// TIA Portal V19 export
FUNCTION "RECIPE" : Void   // FC7, LAD
{ S7_Optimized_Access := 'TRUE' }
// stored: SetENOAutomatically false
BEGIN

REGION Network 1: RINSE 1
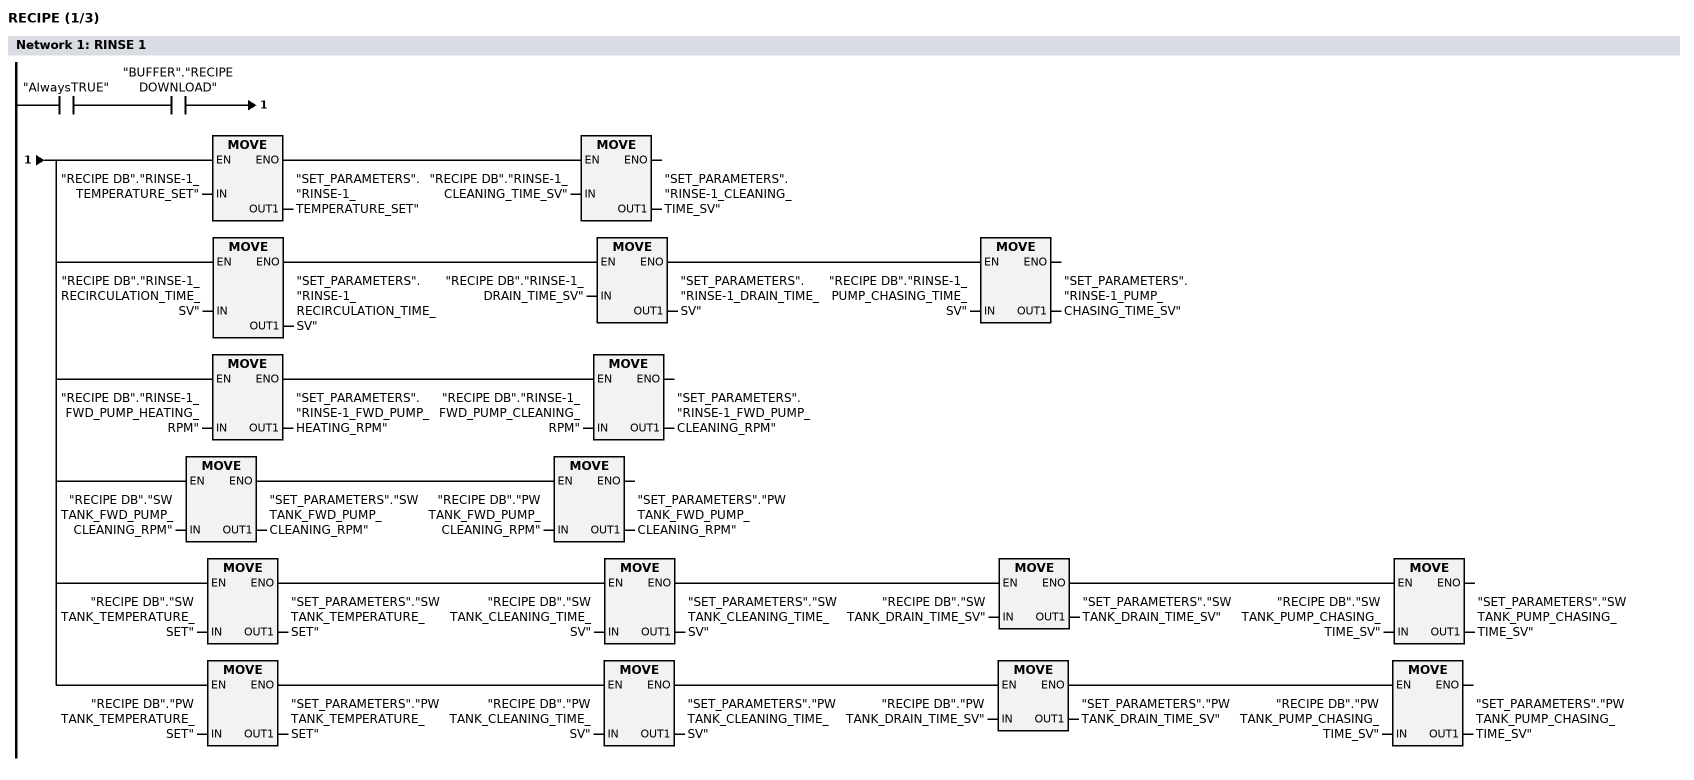
   RUNG wire#powerrail
      Contact( "AlwaysTRUE" )
      Contact( "BUFFER"."RECIPE DOWNLOAD" )
      wire#w1
      Move(in := "RECIPE DB"."RINSE-1_TEMPERATURE_SET", out1 => "SET_PARAMETERS"."RINSE-1_TEMPERATURE_SET")
      Move(in := "RECIPE DB"."RINSE-1_CLEANING_TIME_SV", out1 => "SET_PARAMETERS"."RINSE-1_CLEANING_TIME_SV")
   END_RUNG
   RUNG wire#w1
      Move(in := "RECIPE DB"."RINSE-1_RECIRCULATION_TIME_SV", out1 => "SET_PARAMETERS"."RINSE-1_RECIRCULATION_TIME_SV")
      Move(in := "RECIPE DB"."RINSE-1_DRAIN_TIME_SV", out1 => "SET_PARAMETERS"."RINSE-1_DRAIN_TIME_SV")
      Move(in := "RECIPE DB"."RINSE-1_PUMP_CHASING_TIME_SV", out1 => "SET_PARAMETERS"."RINSE-1_PUMP_CHASING_TIME_SV")
   END_RUNG
   RUNG wire#w1
      Move(in := "RECIPE DB"."RINSE-1_FWD_PUMP_HEATING_RPM", out1 => "SET_PARAMETERS"."RINSE-1_FWD_PUMP_HEATING_RPM")
      Move(in := "RECIPE DB"."RINSE-1_FWD_PUMP_CLEANING_RPM", out1 => "SET_PARAMETERS"."RINSE-1_FWD_PUMP_CLEANING_RPM")
   END_RUNG
   RUNG wire#w1
      Move(in := "RECIPE DB"."SW TANK_FWD_PUMP_CLEANING_RPM", out1 => "SET_PARAMETERS"."SW TANK_FWD_PUMP_CLEANING_RPM")
      Move(in := "RECIPE DB"."PW TANK_FWD_PUMP_CLEANING_RPM", out1 => "SET_PARAMETERS"."PW TANK_FWD_PUMP_CLEANING_RPM")
   END_RUNG
   RUNG wire#w1
      Move(in := "RECIPE DB"."SW TANK_TEMPERATURE_SET", out1 => "SET_PARAMETERS"."SW TANK_TEMPERATURE_SET")
      Move(in := "RECIPE DB"."SW TANK_CLEANING_TIME_SV", out1 => "SET_PARAMETERS"."SW TANK_CLEANING_TIME_SV")
      Move(in := "RECIPE DB"."SW TANK_DRAIN_TIME_SV", out1 => "SET_PARAMETERS"."SW TANK_DRAIN_TIME_SV")
      Move(in := "RECIPE DB"."SW TANK_PUMP_CHASING_TIME_SV", out1 => "SET_PARAMETERS"."SW TANK_PUMP_CHASING_TIME_SV")
   END_RUNG
   RUNG wire#w1
      Move(in := "RECIPE DB"."PW TANK_TEMPERATURE_SET", out1 => "SET_PARAMETERS"."PW TANK_TEMPERATURE_SET")
      Move(in := "RECIPE DB"."PW TANK_CLEANING_TIME_SV", out1 => "SET_PARAMETERS"."PW TANK_CLEANING_TIME_SV")
      Move(in := "RECIPE DB"."PW TANK_DRAIN_TIME_SV", out1 => "SET_PARAMETERS"."PW TANK_DRAIN_TIME_SV")
      Move(in := "RECIPE DB"."PW TANK_PUMP_CHASING_TIME_SV", out1 => "SET_PARAMETERS"."PW TANK_PUMP_CHASING_TIME_SV")
   END_RUNG
   // the same network as SCL:
   IF "AlwaysTRUE" AND "BUFFER"."RECIPE DOWNLOAD" THEN
       "SET_PARAMETERS"."RINSE-1_TEMPERATURE_SET" := "RECIPE DB"."RINSE-1_TEMPERATURE_SET";
       "SET_PARAMETERS"."RINSE-1_CLEANING_TIME_SV" := "RECIPE DB"."RINSE-1_CLEANING_TIME_SV";
       "SET_PARAMETERS"."RINSE-1_RECIRCULATION_TIME_SV" := "RECIPE DB"."RINSE-1_RECIRCULATION_TIME_SV";
       "SET_PARAMETERS"."RINSE-1_DRAIN_TIME_SV" := "RECIPE DB"."RINSE-1_DRAIN_TIME_SV";
       "SET_PARAMETERS"."RINSE-1_PUMP_CHASING_TIME_SV" := "RECIPE DB"."RINSE-1_PUMP_CHASING_TIME_SV";
       "SET_PARAMETERS"."RINSE-1_FWD_PUMP_HEATING_RPM" := "RECIPE DB"."RINSE-1_FWD_PUMP_HEATING_RPM";
       "SET_PARAMETERS"."RINSE-1_FWD_PUMP_CLEANING_RPM" := "RECIPE DB"."RINSE-1_FWD_PUMP_CLEANING_RPM";
       "SET_PARAMETERS"."SW TANK_FWD_PUMP_CLEANING_RPM" := "RECIPE DB"."SW TANK_FWD_PUMP_CLEANING_RPM";
       "SET_PARAMETERS"."PW TANK_FWD_PUMP_CLEANING_RPM" := "RECIPE DB"."PW TANK_FWD_PUMP_CLEANING_RPM";
       "SET_PARAMETERS"."SW TANK_TEMPERATURE_SET" := "RECIPE DB"."SW TANK_TEMPERATURE_SET";
       "SET_PARAMETERS"."SW TANK_CLEANING_TIME_SV" := "RECIPE DB"."SW TANK_CLEANING_TIME_SV";
       "SET_PARAMETERS"."SW TANK_DRAIN_TIME_SV" := "RECIPE DB"."SW TANK_DRAIN_TIME_SV";
       "SET_PARAMETERS"."SW TANK_PUMP_CHASING_TIME_SV" := "RECIPE DB"."SW TANK_PUMP_CHASING_TIME_SV";
       "SET_PARAMETERS"."PW TANK_TEMPERATURE_SET" := "RECIPE DB"."PW TANK_TEMPERATURE_SET";
       "SET_PARAMETERS"."PW TANK_CLEANING_TIME_SV" := "RECIPE DB"."PW TANK_CLEANING_TIME_SV";
       "SET_PARAMETERS"."PW TANK_DRAIN_TIME_SV" := "RECIPE DB"."PW TANK_DRAIN_TIME_SV";
       "SET_PARAMETERS"."PW TANK_PUMP_CHASING_TIME_SV" := "RECIPE DB"."PW TANK_PUMP_CHASING_TIME_SV";
   END_IF;
END_REGION

REGION Network 2: WASH BY ACID / ALKALI
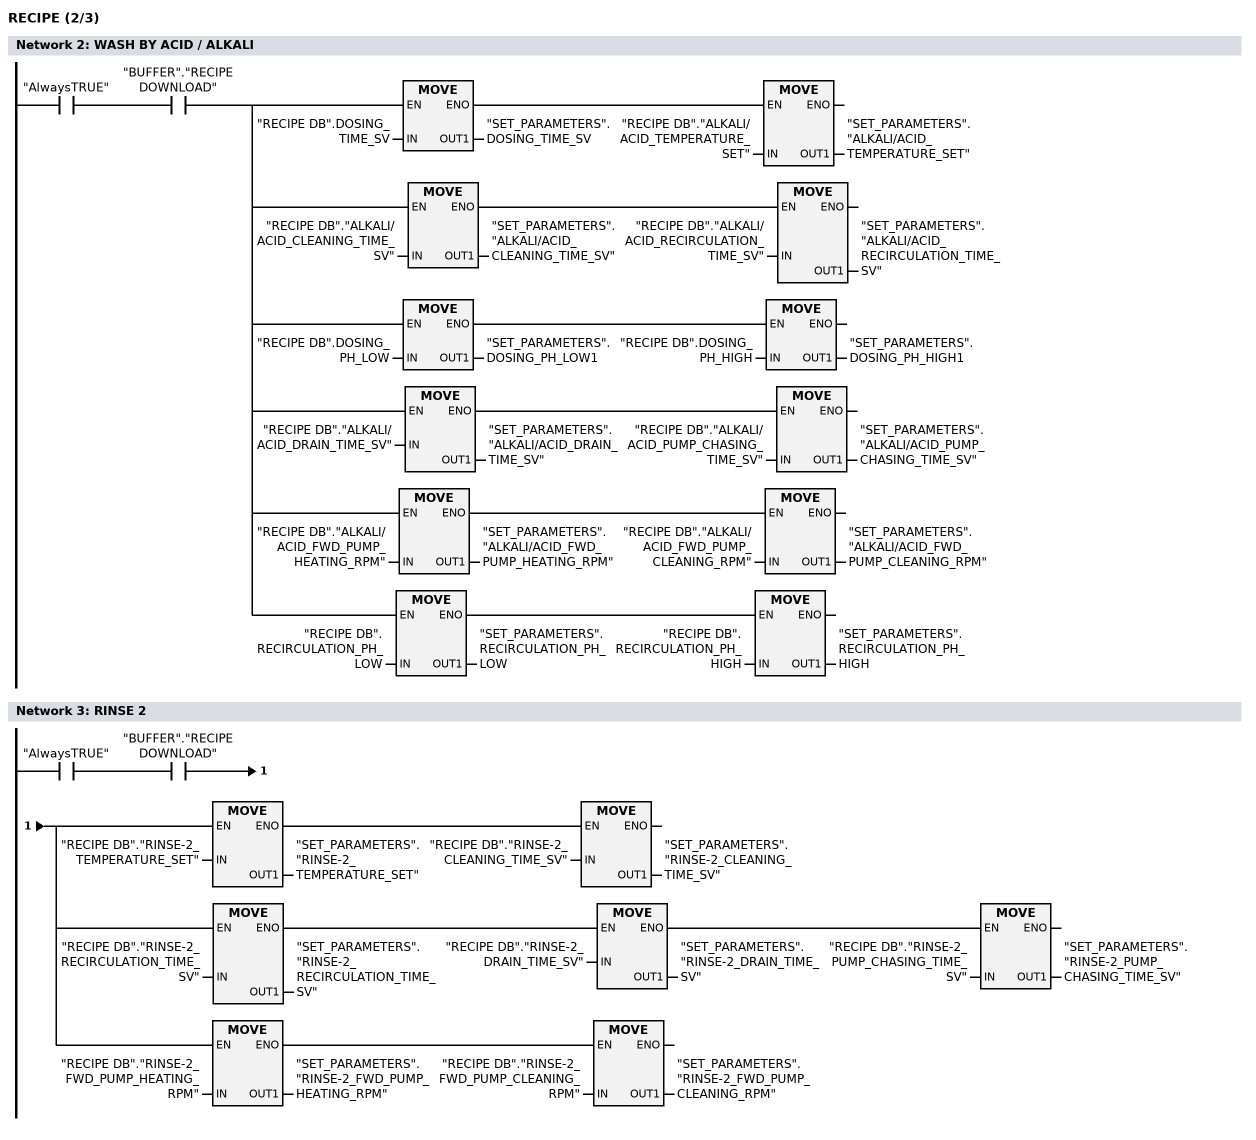
   RUNG wire#powerrail
      Contact( "AlwaysTRUE" )
      Contact( "BUFFER"."RECIPE DOWNLOAD" )
      wire#w1
      Move(in := "RECIPE DB".DOSING_TIME_SV, out1 => "SET_PARAMETERS".DOSING_TIME_SV)
      Move(in := "RECIPE DB"."ALKALI/ACID_TEMPERATURE_SET", out1 => "SET_PARAMETERS"."ALKALI/ACID_TEMPERATURE_SET")
   END_RUNG
   RUNG wire#w1
      Move(in := "RECIPE DB"."ALKALI/ACID_CLEANING_TIME_SV", out1 => "SET_PARAMETERS"."ALKALI/ACID_CLEANING_TIME_SV")
      Move(in := "RECIPE DB"."ALKALI/ACID_RECIRCULATION_TIME_SV", out1 => "SET_PARAMETERS"."ALKALI/ACID_RECIRCULATION_TIME_SV")
   END_RUNG
   RUNG wire#w1
      Move(in := "RECIPE DB".DOSING_PH_LOW, out1 => "SET_PARAMETERS".DOSING_PH_LOW1)
      Move(in := "RECIPE DB".DOSING_PH_HIGH, out1 => "SET_PARAMETERS".DOSING_PH_HIGH1)
   END_RUNG
   RUNG wire#w1
      Move(in := "RECIPE DB"."ALKALI/ACID_DRAIN_TIME_SV", out1 => "SET_PARAMETERS"."ALKALI/ACID_DRAIN_TIME_SV")
      Move(in := "RECIPE DB"."ALKALI/ACID_PUMP_CHASING_TIME_SV", out1 => "SET_PARAMETERS"."ALKALI/ACID_PUMP_CHASING_TIME_SV")
   END_RUNG
   RUNG wire#w1
      Move(in := "RECIPE DB"."ALKALI/ACID_FWD_PUMP_HEATING_RPM", out1 => "SET_PARAMETERS"."ALKALI/ACID_FWD_PUMP_HEATING_RPM")
      Move(in := "RECIPE DB"."ALKALI/ACID_FWD_PUMP_CLEANING_RPM", out1 => "SET_PARAMETERS"."ALKALI/ACID_FWD_PUMP_CLEANING_RPM")
   END_RUNG
   RUNG wire#w1
      Move(in := "RECIPE DB".RECIRCULATION_PH_LOW, out1 => "SET_PARAMETERS".RECIRCULATION_PH_LOW)
      Move(in := "RECIPE DB".RECIRCULATION_PH_HIGH, out1 => "SET_PARAMETERS".RECIRCULATION_PH_HIGH)
   END_RUNG
   // the same network as SCL:
   IF "AlwaysTRUE" AND "BUFFER"."RECIPE DOWNLOAD" THEN
       "SET_PARAMETERS".DOSING_TIME_SV := "RECIPE DB".DOSING_TIME_SV;
       "SET_PARAMETERS"."ALKALI/ACID_TEMPERATURE_SET" := "RECIPE DB"."ALKALI/ACID_TEMPERATURE_SET";
       "SET_PARAMETERS"."ALKALI/ACID_CLEANING_TIME_SV" := "RECIPE DB"."ALKALI/ACID_CLEANING_TIME_SV";
       "SET_PARAMETERS"."ALKALI/ACID_RECIRCULATION_TIME_SV" := "RECIPE DB"."ALKALI/ACID_RECIRCULATION_TIME_SV";
       "SET_PARAMETERS".DOSING_PH_LOW1 := "RECIPE DB".DOSING_PH_LOW;
       "SET_PARAMETERS".DOSING_PH_HIGH1 := "RECIPE DB".DOSING_PH_HIGH;
       "SET_PARAMETERS"."ALKALI/ACID_DRAIN_TIME_SV" := "RECIPE DB"."ALKALI/ACID_DRAIN_TIME_SV";
       "SET_PARAMETERS"."ALKALI/ACID_PUMP_CHASING_TIME_SV" := "RECIPE DB"."ALKALI/ACID_PUMP_CHASING_TIME_SV";
       "SET_PARAMETERS"."ALKALI/ACID_FWD_PUMP_HEATING_RPM" := "RECIPE DB"."ALKALI/ACID_FWD_PUMP_HEATING_RPM";
       "SET_PARAMETERS"."ALKALI/ACID_FWD_PUMP_CLEANING_RPM" := "RECIPE DB"."ALKALI/ACID_FWD_PUMP_CLEANING_RPM";
       "SET_PARAMETERS".RECIRCULATION_PH_LOW := "RECIPE DB".RECIRCULATION_PH_LOW;
       "SET_PARAMETERS".RECIRCULATION_PH_HIGH := "RECIPE DB".RECIRCULATION_PH_HIGH;
   END_IF;
END_REGION

REGION Network 3: RINSE 2
   RUNG wire#powerrail
      Contact( "AlwaysTRUE" )
      Contact( "BUFFER"."RECIPE DOWNLOAD" )
      wire#w1
      Move(in := "RECIPE DB"."RINSE-2_TEMPERATURE_SET", out1 => "SET_PARAMETERS"."RINSE-2_TEMPERATURE_SET")
      Move(in := "RECIPE DB"."RINSE-2_CLEANING_TIME_SV", out1 => "SET_PARAMETERS"."RINSE-2_CLEANING_TIME_SV")
   END_RUNG
   RUNG wire#w1
      Move(in := "RECIPE DB"."RINSE-2_RECIRCULATION_TIME_SV", out1 => "SET_PARAMETERS"."RINSE-2_RECIRCULATION_TIME_SV")
      Move(in := "RECIPE DB"."RINSE-2_DRAIN_TIME_SV", out1 => "SET_PARAMETERS"."RINSE-2_DRAIN_TIME_SV")
      Move(in := "RECIPE DB"."RINSE-2_PUMP_CHASING_TIME_SV", out1 => "SET_PARAMETERS"."RINSE-2_PUMP_CHASING_TIME_SV")
   END_RUNG
   RUNG wire#w1
      Move(in := "RECIPE DB"."RINSE-2_FWD_PUMP_HEATING_RPM", out1 => "SET_PARAMETERS"."RINSE-2_FWD_PUMP_HEATING_RPM")
      Move(in := "RECIPE DB"."RINSE-2_FWD_PUMP_CLEANING_RPM", out1 => "SET_PARAMETERS"."RINSE-2_FWD_PUMP_CLEANING_RPM")
   END_RUNG
   // the same network as SCL:
   IF "AlwaysTRUE" AND "BUFFER"."RECIPE DOWNLOAD" THEN
       "SET_PARAMETERS"."RINSE-2_TEMPERATURE_SET" := "RECIPE DB"."RINSE-2_TEMPERATURE_SET";
       "SET_PARAMETERS"."RINSE-2_CLEANING_TIME_SV" := "RECIPE DB"."RINSE-2_CLEANING_TIME_SV";
       "SET_PARAMETERS"."RINSE-2_RECIRCULATION_TIME_SV" := "RECIPE DB"."RINSE-2_RECIRCULATION_TIME_SV";
       "SET_PARAMETERS"."RINSE-2_DRAIN_TIME_SV" := "RECIPE DB"."RINSE-2_DRAIN_TIME_SV";
       "SET_PARAMETERS"."RINSE-2_PUMP_CHASING_TIME_SV" := "RECIPE DB"."RINSE-2_PUMP_CHASING_TIME_SV";
       "SET_PARAMETERS"."RINSE-2_FWD_PUMP_HEATING_RPM" := "RECIPE DB"."RINSE-2_FWD_PUMP_HEATING_RPM";
       "SET_PARAMETERS"."RINSE-2_FWD_PUMP_CLEANING_RPM" := "RECIPE DB"."RINSE-2_FWD_PUMP_CLEANING_RPM";
   END_IF;
END_REGION

REGION Network 4: RINSE 3 (FIANL_RINSE-1)
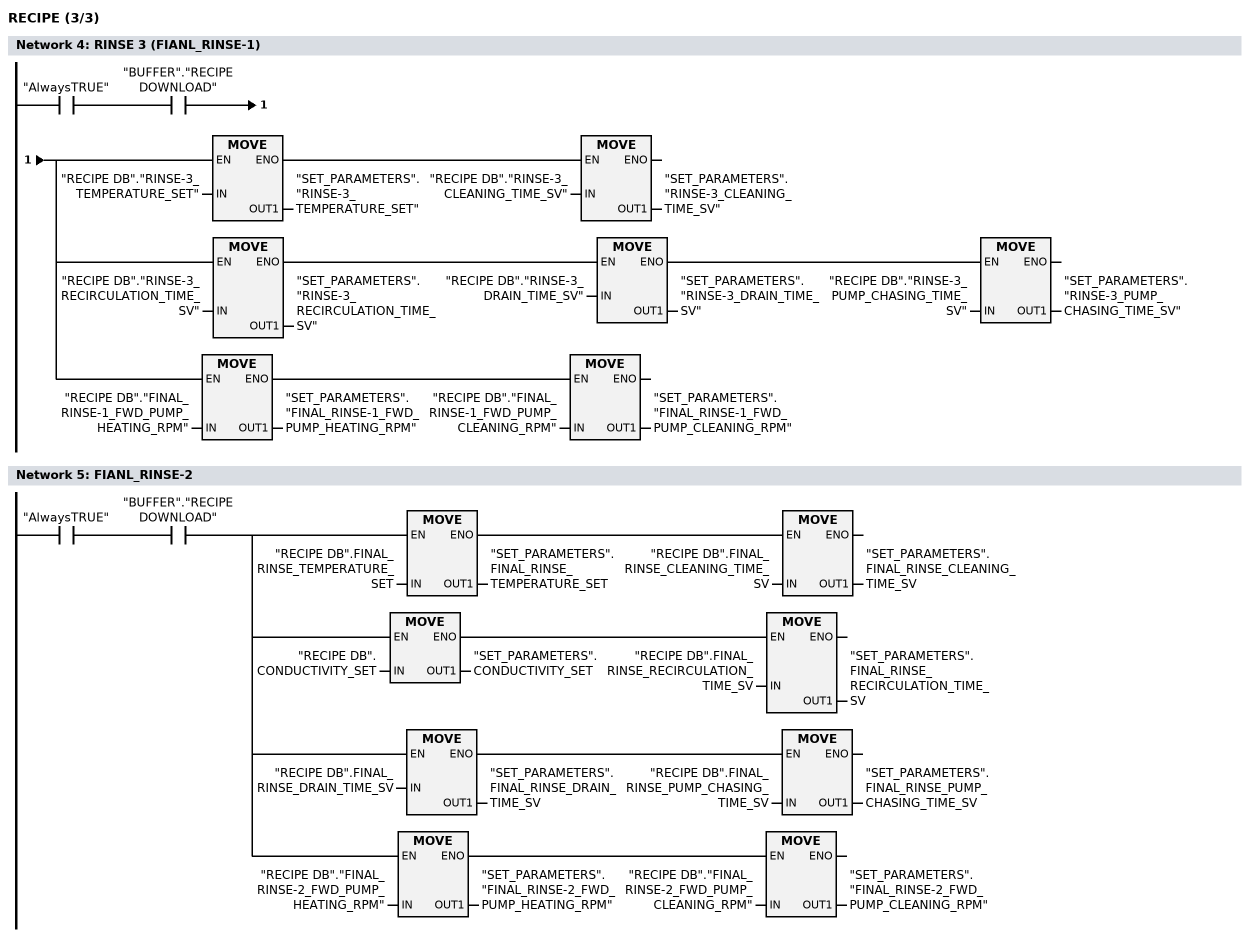
   RUNG wire#powerrail
      Contact( "AlwaysTRUE" )
      Contact( "BUFFER"."RECIPE DOWNLOAD" )
      wire#w1
      Move(in := "RECIPE DB"."RINSE-3_TEMPERATURE_SET", out1 => "SET_PARAMETERS"."RINSE-3_TEMPERATURE_SET")
      Move(in := "RECIPE DB"."RINSE-3_CLEANING_TIME_SV", out1 => "SET_PARAMETERS"."RINSE-3_CLEANING_TIME_SV")
   END_RUNG
   RUNG wire#w1
      Move(in := "RECIPE DB"."RINSE-3_RECIRCULATION_TIME_SV", out1 => "SET_PARAMETERS"."RINSE-3_RECIRCULATION_TIME_SV")
      Move(in := "RECIPE DB"."RINSE-3_DRAIN_TIME_SV", out1 => "SET_PARAMETERS"."RINSE-3_DRAIN_TIME_SV")
      Move(in := "RECIPE DB"."RINSE-3_PUMP_CHASING_TIME_SV", out1 => "SET_PARAMETERS"."RINSE-3_PUMP_CHASING_TIME_SV")
   END_RUNG
   RUNG wire#w1
      Move(in := "RECIPE DB"."FINAL_RINSE-1_FWD_PUMP_HEATING_RPM", out1 => "SET_PARAMETERS"."FINAL_RINSE-1_FWD_PUMP_HEATING_RPM")
      Move(in := "RECIPE DB"."FINAL_RINSE-1_FWD_PUMP_CLEANING_RPM", out1 => "SET_PARAMETERS"."FINAL_RINSE-1_FWD_PUMP_CLEANING_RPM")
   END_RUNG
   // the same network as SCL:
   IF "AlwaysTRUE" AND "BUFFER"."RECIPE DOWNLOAD" THEN
       "SET_PARAMETERS"."RINSE-3_TEMPERATURE_SET" := "RECIPE DB"."RINSE-3_TEMPERATURE_SET";
       "SET_PARAMETERS"."RINSE-3_CLEANING_TIME_SV" := "RECIPE DB"."RINSE-3_CLEANING_TIME_SV";
       "SET_PARAMETERS"."RINSE-3_RECIRCULATION_TIME_SV" := "RECIPE DB"."RINSE-3_RECIRCULATION_TIME_SV";
       "SET_PARAMETERS"."RINSE-3_DRAIN_TIME_SV" := "RECIPE DB"."RINSE-3_DRAIN_TIME_SV";
       "SET_PARAMETERS"."RINSE-3_PUMP_CHASING_TIME_SV" := "RECIPE DB"."RINSE-3_PUMP_CHASING_TIME_SV";
       "SET_PARAMETERS"."FINAL_RINSE-1_FWD_PUMP_HEATING_RPM" := "RECIPE DB"."FINAL_RINSE-1_FWD_PUMP_HEATING_RPM";
       "SET_PARAMETERS"."FINAL_RINSE-1_FWD_PUMP_CLEANING_RPM" := "RECIPE DB"."FINAL_RINSE-1_FWD_PUMP_CLEANING_RPM";
   END_IF;
END_REGION

REGION Network 5: FIANL_RINSE-2
   RUNG wire#powerrail
      Contact( "AlwaysTRUE" )
      Contact( "BUFFER"."RECIPE DOWNLOAD" )
      wire#w1
      Move(in := "RECIPE DB".FINAL_RINSE_TEMPERATURE_SET, out1 => "SET_PARAMETERS".FINAL_RINSE_TEMPERATURE_SET)
      Move(in := "RECIPE DB".FINAL_RINSE_CLEANING_TIME_SV, out1 => "SET_PARAMETERS".FINAL_RINSE_CLEANING_TIME_SV)
   END_RUNG
   RUNG wire#w1
      Move(in := "RECIPE DB".CONDUCTIVITY_SET, out1 => "SET_PARAMETERS".CONDUCTIVITY_SET)
      Move(in := "RECIPE DB".FINAL_RINSE_RECIRCULATION_TIME_SV, out1 => "SET_PARAMETERS".FINAL_RINSE_RECIRCULATION_TIME_SV)
   END_RUNG
   RUNG wire#w1
      Move(in := "RECIPE DB".FINAL_RINSE_DRAIN_TIME_SV, out1 => "SET_PARAMETERS".FINAL_RINSE_DRAIN_TIME_SV)
      Move(in := "RECIPE DB".FINAL_RINSE_PUMP_CHASING_TIME_SV, out1 => "SET_PARAMETERS".FINAL_RINSE_PUMP_CHASING_TIME_SV)
   END_RUNG
   RUNG wire#w1
      Move(in := "RECIPE DB"."FINAL_RINSE-2_FWD_PUMP_HEATING_RPM", out1 => "SET_PARAMETERS"."FINAL_RINSE-2_FWD_PUMP_HEATING_RPM")
      Move(in := "RECIPE DB"."FINAL_RINSE-2_FWD_PUMP_CLEANING_RPM", out1 => "SET_PARAMETERS"."FINAL_RINSE-2_FWD_PUMP_CLEANING_RPM")
   END_RUNG
   // the same network as SCL:
   IF "AlwaysTRUE" AND "BUFFER"."RECIPE DOWNLOAD" THEN
       "SET_PARAMETERS".FINAL_RINSE_TEMPERATURE_SET := "RECIPE DB".FINAL_RINSE_TEMPERATURE_SET;
       "SET_PARAMETERS".FINAL_RINSE_CLEANING_TIME_SV := "RECIPE DB".FINAL_RINSE_CLEANING_TIME_SV;
       "SET_PARAMETERS".CONDUCTIVITY_SET := "RECIPE DB".CONDUCTIVITY_SET;
       "SET_PARAMETERS".FINAL_RINSE_RECIRCULATION_TIME_SV := "RECIPE DB".FINAL_RINSE_RECIRCULATION_TIME_SV;
       "SET_PARAMETERS".FINAL_RINSE_DRAIN_TIME_SV := "RECIPE DB".FINAL_RINSE_DRAIN_TIME_SV;
       "SET_PARAMETERS".FINAL_RINSE_PUMP_CHASING_TIME_SV := "RECIPE DB".FINAL_RINSE_PUMP_CHASING_TIME_SV;
       "SET_PARAMETERS"."FINAL_RINSE-2_FWD_PUMP_HEATING_RPM" := "RECIPE DB"."FINAL_RINSE-2_FWD_PUMP_HEATING_RPM";
       "SET_PARAMETERS"."FINAL_RINSE-2_FWD_PUMP_CLEANING_RPM" := "RECIPE DB"."FINAL_RINSE-2_FWD_PUMP_CLEANING_RPM";
   END_IF;
END_REGION
END_FUNCTION
